PROGRAM P_Demo_INT64_TO_LREAL
VAR
    liTorqueInt  : T_LARGE_INTEGER;; // 有符号 64 位扭矩积分
    lrTorqueDisp : LREAL;; // HMI 显示
    bConvert     : BOOL;
END_VAR

// ============================================================
// Tc2_Utilities.INT64_TO_LREAL 演示程序（FUNCTION，单周期触发）
// ============================================================
// 场景：把 64 位有符号扭矩积分（可正可负）转 LREAL 在 HMI 显示。
// 价值：替代手写有符号双倍长转浮点；一行调用。
// 验证步骤：
//   1. 把本 PROGRAM 加到 PlcTask 调用列表
//   2. 编译 + 登录
//   3. 在线把 b... 触发位置 TRUE 一个周期
//   4. 观察输出变量是否符合期望
// ============================================================

IF bConvert THEN
    lrTorqueDisp := INT64_TO_LREAL(liTorqueInt);
    bConvert := FALSE;
END_IF;

END_PROGRAM

(* stored: Version 1.1.0.1, ProductVersion 3.1.4024.5
   POU P_Demo_INT64_TO_LREAL: Id {fc1a4c00-470c-5979-adf2-3ee033929c16}, SpecialFunc None *)
